{attribute 'qualified_only'}
{attribute 'strict'}
TYPE E_MachineMode :
(
	Manual := 0,
	Auto
);
END_TYPE

(* stored: Version 1.1.0.1, ProductVersion 3.1.4024.16
   DUT E_MachineMode: Id {0425caa7-0fca-467f-b7a7-2cece76509d0} *)
